// TIA Portal V20 export
DATA_BLOCK "DB_Alarm"   // DB17
// stored: Access Published, MemoryReserve 100, Namespace Global
   VAR
      "word" : Struct
         Line : Struct
            A1 : Struct
               Conveyor : Array[_.gMinA1.._.gMaxA1] of Word;
            END_STRUCT;
            B1 : Struct
               Conveyor : Array[_.gMinB1.._.gMaxB1] of Word;
            END_STRUCT;
            C1 : Struct
               Conveyor : Array[_.gMinC1.._.gMaxC1] of Word;
            END_STRUCT;
            D1 : Struct
               Conveyor : Array[_.gMinD1.._.gMaxD1] of Word;
            END_STRUCT;
         END_STRUCT;
      END_STRUCT;
      HardDiag : Struct
         ASi : Word;
         Nord : Word;
      END_STRUCT;
   END_VAR
BEGIN
END_DATA_BLOCK
